///Automatically generated by BoxConfigurator 
TYPE E_GroupNumber :
(
	G_BEGIN_GROUP,
	G_SG_001,
	G_SG_002,
	G_END_GROUP
);
END_TYPE

(* stored: Version 1.1.0.1, ProductVersion 3.1.4024.9
   DUT E_GroupNumber: Id {9addbec1-7b3d-4d44-b9ce-b3dde73fa330} *)
